Universal Robots PolyScope program: impedance intro.urp

Program impedance intro new (createdIn=3.2.19293.0 lastSavedIn=3.5.0.10584 directory=/programs installation=default robotSerialNumber=2016352577)
Calibrated DH parameters: a=[0.000176, -0.30042, -0.37922, 0.000042, 0.000063, 0]; d=[0.089415, 194.329143, -181.748083, -12.470753, 0.09493, 0.082587]; alpha=[1.570535, -0.00155, 0.008062, 1.570056, -1.571015, 0]; deltaTheta=[-0.000017, -0.786835, 1.048193, -0.261404, -0.000054, -0.000059]
BeforeStart
  stop_timer := False
  timer := 0
Robot Program (runOnlyOnce=false motionType=MoveJ speed=1.047198 acceleration=1.396263 useActiveTCP=false)
  Loop Forever
    Script file /programs/usbdisk_0/impedance intro code.txt_bak
      | #    This program is free software: you can redistribute it and/or modify
      | #    it under the terms of the GNU General Public License as published by
      | #    the Free Software Foundation, either version 3 of the License, or
      | #    (at your option) any later version.
      | #
      | #    This program is distributed in the hope that it will be useful,
      | #    but WITHOUT ANY WARRANTY; without even the implied warranty of
      | #    MERCHANTABILITY or FITNESS FOR A PARTICULAR PURPOSE.  See the
      | #    GNU General Public License for more details.
      | #
      | #    You should have received a copy of the GNU General Public License
      | #    along with this program.  If not, see <https://www.gnu.org/licenses/>.
      | 
      | def Prog1():
      | 
      | 	# Grab Current Position as Start Position
      | 	global start_pose = get_actual_tcp_pose()
      | 
      | 	#Initialize some global variables
      | 	global x_start = start_pose[0]
      | 	global y_start = start_pose[1]
      | 	global z_start = start_pose[2]
      | 	global Rx_start = start_pose[3]
      | 	global Ry_start = start_pose[4]
      | 	global Rz_start = start_pose[5]
      | 	global vx = 0.0
      | 	global vy = 0.0
      | 	global vz = 0.0
      | 	global dt = 0.0
      | 	global Fx_low = 0.0
      | 	global Fy_low = 0.0
      | 	global Fz_low = 0.0
      | 	global x_actual = 0.0
      | 	global y_actual = 0.0
      | 	global z_actual = 0.0
      | 	stop_timer = True
      | 
      | 	#Initialize variables
      | 	x_new = x_start
      | 	y_new = y_start
      | 	z_new = z_start
      | 
      | 	#Spring constants in N/m
      | 	K_x = 100.0
      | 	K_y = 100.0
      | 	K_z = 100.0
      | 
      | 	#Damping coefficients in N/(m/s)
      | 	B_x = 8.94
      | 	B_y = 8.94
      | 	B_z = 8.94
      | 
      | 	#Masses in kg
      | 	M_x = .2
      | 	M_y = .2
      | 	M_z = .2
      | 
      | 	Fx_low = 0.0
      | 	Fy_low = 0.0
      | 	Fz_low = 0.0
      | 	global Fx_bias = 0.0
      | 	global Fy_bias = 0.0
      | 	global Fz_bias = 0.0
      | 
      | 	#Desired force offset (e.g. to apply a force to an object)
      | 	Fdx = 0.0
      | 	Fdy = 0.0
      | 	Fdz = 0.0
      | 
      | 	#Average the force sensor readings for one second to find a force bias vector in the end effector frame
      | 	i=0
      | 	while i<125:
      | 		Fx_bias = Fx_bias + .008 * Fx
      | 		Fy_bias = Fy_bias + .008 * Fy
      | 		Fz_bias = Fz_bias + .008 * Fz
      | 		sync()
      | 		i=i+1
      | 	end
      | 
      | 	#Use Rodrigues' rotation formula to rotate the force bias vector into the base frame
      | 	mag_k = sqrt(Rx_start*Rx_start + Ry_start*Ry_start + Rz_start*Rz_start)
      | 	theta = mag_k
      | 	k_hat = [Rx_start/mag_k, Ry_start/mag_k, Rz_start/mag_k]
      | 	v = [Fx_bias, Fy_bias, Fz_bias]
      | 	vctheta = [v[0]*cos(theta), v[1]*cos(theta), v[2]*cos(theta)]
      | 	kcrossv = [k_hat[1]*v[2] - k_hat[2]*v[1], k_hat[2]*v[0] - k_hat[0]*v[2], k_hat[0]*v[1] - k_hat[1]*v[0]]
      | 	kcrossv_st = [sin(theta)*kcrossv[0], sin(theta)*kcrossv[1], sin(theta)*kcrossv[2]]
      | 	kdotv = k_hat[0]*v[0] + k_hat[1]*v[1] + k_hat[2]*v[2]
      | 	v_rot = [0.0, 0.0, 0.0]
      | 	v_rot[0] = vctheta[0] + kcrossv_st[0] + k_hat[0]*kdotv*(1-cos(theta))
      | 	v_rot[1] = vctheta[1] + kcrossv_st[1] + k_hat[1]*kdotv*(1-cos(theta))
      | 	v_rot[2] = vctheta[2] + kcrossv_st[2] + k_hat[2]*kdotv*(1-cos(theta))
      | 	Fx_bias = v_rot[0]
      | 	Fy_bias = v_rot[1]
      | 	Fz_bias = v_rot[2]
      | 
      | 
      | 	#Get the robot's starting pose
      | 	global new_pose = get_actual_tcp_pose()
      | 	global current_pose = get_actual_tcp_pose()
      | 	global x_current = current_pose[0]
      | 	global y_current = current_pose[1]
      | 	global z_current = current_pose[2]
      | 	global Rx_current = current_pose[3]
      | 	global Ry_current = current_pose[4]
      | 	global Rz_current = current_pose[5]
      | 
      | 	global x_error = 0.0
      | 	global y_error = 0.0
      | 	global z_error = 0.0
      | 
      | 
      | 	i = 0
      | 	last_time = timer - .008
      | 	xd = x_current
      | 	yd = y_current
      | 	zd = z_current
      | 	dt = .008
      | 
      | 	#Enter the main loop
      | 	while i < 1:
      | 		#Compute a desired trajectory
      | 		#In this case, it goes back to the start position
      | 		xdnew = x_start
      | 		ydnew = y_start
      | 		zdnew = z_start
      | 
      | 		#Avoid dividing by zero
      | 		if dt  == 0.0:
      | 			dt = 0.001
      | 		end
      | 
      | 		#Differentiate desired position to find desired velocity
      | 		vxd = 1.0 / dt * (xdnew - xd)
      | 		vyd = 1.0 / dt * (ydnew - yd)
      | 		vzd = 1.0 / dt * (zdnew - zd)
      | 		xd = xdnew
      | 		yd = ydnew
      | 		zd = zdnew
      | 
      | 		#Read the pose of the end effector
      | 		pose_actual = get_actual_tcp_pose()
      | 		x_actual = pose_actual[0]
      | 		y_actual = pose_actual[1]
      | 		z_actual = pose_actual[2]
      | 		Rx_actual = pose_actual[3]
      | 		Ry_actual = pose_actual[4]
      | 		Rz_actual = pose_actual[5]
      | 
      | 		#Monitor the end effector's distance from the commanded position
      | 		x_error = x_current - x_actual
      | 		y_error = y_current - y_actual
      | 		z_error = z_current - z_actual
      | 
      | 		global new_pose = current_pose
      | 
      | 		#Use a low pass filter on incoming force measurements
      | 		#global Fx_low = .062*Fx + (1.0-.062)*Fx_low
      | 		#global Fy_low = .062*Fy + (1.0-.062)*Fy_low
      | 		#global Fz_low = .062*Fz + (1.0-.062)*Fz_low
      | 
      | 		#Use Rodrigues' rotation formula to rotate the low pass filtered force measurements into the base frame
      | 		mag_k = sqrt(Rx_actual * Rx_actual + Ry_actual * Ry_actual + Rz_actual * Rz_actual)
      | 		theta = mag_k
      | 		k_hat = [Rx_actual / mag_k, Ry_actual / mag_k, Rz_actual / mag_k]
      | 		#v = [Fx_low, Fy_low, Fz_low]
      | 		v = [Fx, Fy, Fz]
      | 		vctheta = [v[0] * cos(theta), v[1] * cos(theta), v[2] * cos(theta)]
      | 		kcrossv = [k_hat[1] * v[2] - k_hat[2] * v[1], k_hat[2] * v[0] - k_hat[0] * v[2], k_hat[0] * v[1] - k_hat[1] * v[0]]
      | 		kcrossv_st = [sin(theta) * kcrossv[0], sin(theta) * kcrossv[1], sin(theta) * kcrossv[2]]
      | 		kdotv = k_hat[0] * v[0] + k_hat[1] * v[1] + k_hat[2] * v[2]
      | 		v_rot = [0.0, 0.0, 0.0]
      | 		v_rot[0] = vctheta[0] + kcrossv_st[0] + k_hat[0] * kdotv * (1 - cos(theta))
      | 		v_rot[1] = vctheta[1] + kcrossv_st[1] + k_hat[1] * kdotv * (1 - cos(theta))
      | 		v_rot[2] = vctheta[2] + kcrossv_st[2] + k_hat[2] * kdotv * (1 - cos(theta))
      | 		corrected_forces = p[v_rot[0], v_rot[1], v_rot[2], 0,0,0]
      | 
      | 
      | 		#Correct the forces by subtracting the force bias
      | 		c_Fx_low = corrected_forces[0] - Fx_bias
      | 		c_Fy_low = corrected_forces[1] - Fy_bias
      | 		c_Fz_low = corrected_forces[2] - Fz_bias
      | 
      | 		#Find the resulting acceleration given the forces on the end effector
      | 		#The acceleration is determined based on the admittance control law
      | 		a_x = 1.0/M_x * (K_x * (xd - x_current) - B_x * (vx - vxd) + c_Fx_low + Fdx)
      | 		a_y = 1.0/M_y * (K_y * (yd - y_current) - B_y * (vy - vyd) + c_Fy_low + Fdy)
      | 		a_z = 1.0/M_z * (K_z * (zd - z_current) - B_z * (vz - vzd) + c_Fz_low + Fdz)
      | 
      | 		dt = timer - last_time
      | 
      | 		#Integrate the acceleration and velocity to get position
      | 		x_new = x_current + vx*dt + .5*a_x*dt*dt
      | 		y_new = y_current + vy*dt + .5*a_y*dt*dt
      | 		z_new = z_current + vz*dt + .5*a_z*dt*dt
      | 
      | 		x_current = x_new
      | 		y_current = y_new
      | 		z_current = z_new
      | 
      | 		#Keep using the starting rotation
      | 		Rx_current = Rx_start
      | 		Ry_current = Ry_start
      | 		Rz_current = Rz_start
      | 
      | 		#Integrate acceleration to get velocity
      | 		vx = vx + a_x * dt
      | 		vy = vy + a_y * dt
      | 		vz = vz + a_z * dt
      | 
      | 		#Construct the new robot pose
      | 		new_pose[0] = x_current
      | 		new_pose[1] = y_current
      | 		new_pose[2] = z_current
      | 		new_pose[3] = Rx_current
      | 		new_pose[4] = Ry_current
      | 		new_pose[5] = Rz_current
      | 
      | 		#Send the resulting pose to the robot
      | 		servoj(get_inverse_kin(new_pose), lookahead_time=0.2, gain=100)
      | 		last_time = timer
      | 		sleep(.001)
      | 	end
      | end
      | -
      | Prog1()
    Wait Sleep waitTime=0.01
    MoveJ speed 60 deg/s, acceleration 80 deg/s^2 (useActiveTCP=false)
      Waypoint Waypoint_7: TCP in base x=-33.181 y=-370.146 z=538.529 mm, rx=-2.2219 ry=-2.2209 rz=-0.0009 rad; joints [-77.778, -74.533, -87.527, -107.945, 90.387, 102.035] deg
Thread Thread_1 (runOnlyOnce=false trackProgramExecution=false)
  sensor_data := socket_read_ascii_float(6,"stream")
  If sensor_data[0] ≥6
    Fx := sensor_data[1]   [initializeExpression=0.0]
    Fy := sensor_data[2]   [initializeExpression=0.0]
    Fz := sensor_data[3]   [initializeExpression=0.0]
    Mx := sensor_data[4]   [initializeExpression=0.0]
    My := sensor_data[5]   [initializeExpression=0.0]
    Mz := sensor_data[6]   [initializeExpression=0.0]
  Else 
    Fx := 0.0
    Fy := 0.0
    Fz := 0.0
    Mx := 0.0
    My := 0.0
    Mz := 0.0
Thread Thread_2 (runOnlyOnce=false trackProgramExecution=false)
  If stop_timer ≟ True
    Script: timer = timer +.008
  Else 
    Script: timer =0
  Wait Sleep waitTime=0.008
